PROGRAM MAIN
VAR
END_VAR

END_PROGRAM

(* stored: Version 1.1.0.1
   POU MAIN: Id {d32cfe5f-db53-4421-8d8c-1553de2c8f1c} *)
